SUBAPPLICATION Uebung_006a3 (* SR und T-Flip-Flop mit 3x IE *)
  (* Standard: 61499-2; Description: Copyright (c) 2023 Meisterschulen am Ostbahnhof This program and the accompanying materials are made available under the terms of the Eclipse Public License 2.0 which is available at https://www.eclipse.org/legal/epl-2.0/ SPDX-License-Identifier: EPL-2.0 *)
  (* Version 1.0, 2023-10-23, Franz Höpfinger, Meisterschulen am Ostbahnhof *)
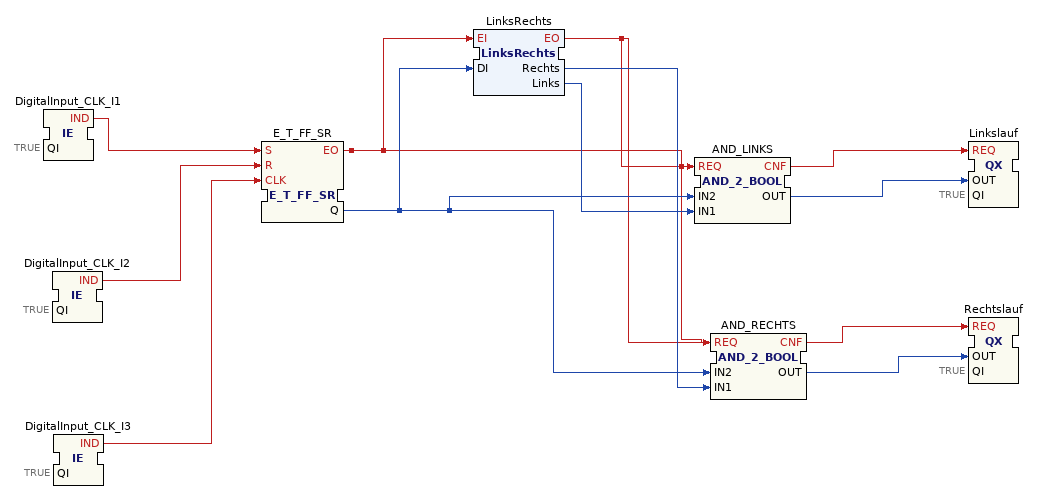
  FBS
    DigitalInput_CLK_I1 : IE(QI := TRUE);
    DigitalInput_CLK_I2 : IE(QI := TRUE);
    E_T_FF_SR : E_T_FF_SR;
    DigitalInput_CLK_I3 : IE(QI := TRUE);
    AND_LINKS : AND_2_BOOL;
    Rechtslauf : QX(QI := TRUE);
    Linkslauf : QX(QI := TRUE);
    AND_RECHTS : AND_2_BOOL;
  END_FBS
  SUBAPPS
    LinksRechts : LinksRechts;
  END_SUBAPPS
  EVENT_CONNECTIONS
    DigitalInput_CLK_I1.IND TO E_T_FF_SR.S;
    DigitalInput_CLK_I2.IND TO E_T_FF_SR.R;
    DigitalInput_CLK_I3.IND TO E_T_FF_SR.CLK;
    AND_RECHTS.CNF TO Rechtslauf.REQ;
    AND_LINKS.CNF TO Linkslauf.REQ;
    E_T_FF_SR.EO TO LinksRechts.EI;
    LinksRechts.EO TO AND_LINKS.REQ;
    LinksRechts.EO TO AND_RECHTS.REQ;
    E_T_FF_SR.EO TO AND_LINKS.REQ;
    E_T_FF_SR.EO TO AND_RECHTS.REQ;
  END_CONNECTIONS
  DATA_CONNECTIONS
    AND_LINKS.OUT TO Linkslauf.OUT;
    E_T_FF_SR.Q TO AND_RECHTS.IN2;
    AND_RECHTS.OUT TO Rechtslauf.OUT;
    E_T_FF_SR.Q TO AND_LINKS.IN2;
    LinksRechts.Rechts TO AND_RECHTS.IN1;
    E_T_FF_SR.Q TO LinksRechts.DI;
    LinksRechts.Links TO AND_LINKS.IN1;
  END_CONNECTIONS
END_SUBAPPLICATION
